Yaskawa INFORM job: pipe_bracket_planes_program.JBI

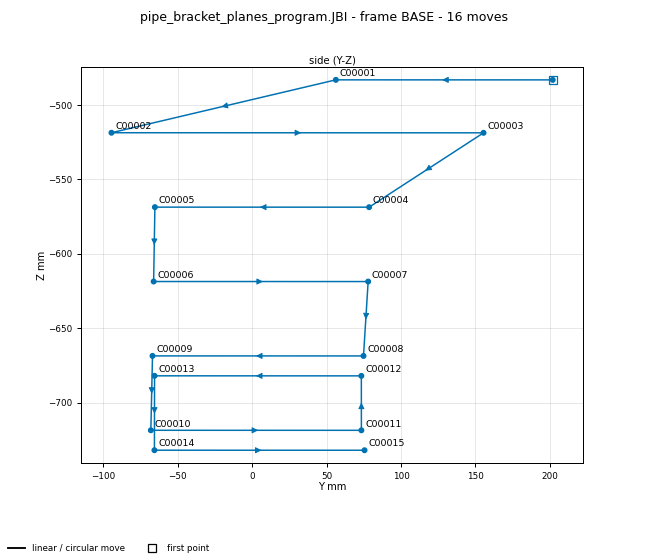
[picture p0: tool path of pipe_bracket_planes_program.JBI in frame BASE, 16 of 18 moves have a stored position in this frame; points joined in program order, loops and branches not executed]
/JOB
//NAME pipe_bracket_planes_program
//POS
///NPOS 16,0,16,0,0,0
///TOOL 0
///POSTYPE BASE
///RECTAN
///RCONF 0,0,0,0,0,0,0,0,0,0,0,0,0,0,0,0,0,0,0,0,0,0,0,0
C00000=1834.327603,202.011474,-483.085613,175.000000,-89.833827,-5.000000
C00001=1836.662464,56.221308,-483.062243,175.000000,-89.833827,-5.000000
C00002=1832.425068,-94.614603,-518.609426,175.000000,-89.833827,-5.000000
C00003=1835.130352,155.502118,-518.668983,175.000000,-89.833827,-5.000000
C00004=1835.789645,78.580596,-568.655204,175.000000,-89.833827,-5.000000
C00005=1835.729919,-65.419986,-568.625259,175.000000,-89.833827,-5.000000
C00006=1836.156481,-66.265346,-618.626533,175.000000,-89.833827,-5.000000
C00007=1834.941053,77.929122,-618.652819,175.000000,-89.833827,-5.000000
C00008=1834.281641,74.809946,-668.650473,175.000000,-89.833827,-5.000000
C00009=1836.578720,-67.033014,-668.627810,175.000000,-89.833827,-5.000000
C00010=1836.499184,-68.140067,-718.627562,175.000000,-89.833827,-5.000000
C00011=1834.131604,73.389504,-718.649955,175.000000,-89.833827,-5.000000
C00012=1834.171210,73.355017,-682.047734,175.000000,-89.833827,-5.000000
C00013=1834.605189,-65.652126,-682.020254,175.000000,-89.833827,-5.000000
C00014=1835.790177,-65.735127,-732.023885,175.000000,-89.833827,-5.000000
C00015=1834.295422,75.507072,-732.048751,180.000000,-60.000000,0.000000
///POSTYPE PULSE
///PULSE
EC00000=192512.0
EC00001=192512.0
EC00002=192512.0
EC00003=192512.0
EC00004=192512.0
EC00005=192512.0
EC00006=192512.0
EC00007=192512.0
EC00008=192512.0
EC00009=192512.0
EC00010=192512.0
EC00011=192512.0
EC00012=192512.0
EC00013=192512.0
EC00014=192512.0
EC00015=192512.0
//INST
///DATE 2023/08/16 18:21
///ATTR SC,RW,RJ
////FRAME BASE
///GROUP1 RB1,ST1
NOP
MOVJ P009 EX000 VJ=15.00
MOVJ C00000 EC00000 VJ=15.0
CALL JOB:SPYON
MOVL C00001 EC00001 V=150.0
MOVL C00002 EC00002 V=150.0
MOVL C00003 EC00003 V=150.0
MOVL C00004 EC00004 V=150.0
MOVL C00005 EC00005 V=150.0
MOVL C00006 EC00006 V=150.0
MOVL C00007 EC00007 V=150.0
MOVL C00008 EC00008 V=150.0
MOVL C00009 EC00009 V=150.0
MOVL C00010 EC00010 V=150.0
MOVL C00011 EC00011 V=150.0
MOVL C00012 EC00012 V=150.0
MOVL C00013 EC00013 V=150.0
MOVL C00014 EC00014 V=150.0
MOVL C00015 EC00015 V=150.0
CALL JOB:SPYOF
MOVJ P009 VJ=15.00
END
